TYPE ST_EmptyStruct :
STRUCT
END_STRUCT
END_TYPE

(* stored: Version 1.1.0.1, ProductVersion 3.1.4024.12
   DUT ST_EmptyStruct: Id {eb9d06b7-5e35-41f3-b199-e2e03ad8220f} *)
